SUBAPPLICATION Uebung_016 (* Subapplication Type *)
  (* Standard: 61499-2 *)
  (* Version 1.0, 2023-10-23, franz *)
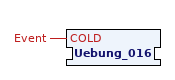
  EVENT_INPUT
    COLD;
  END_EVENT
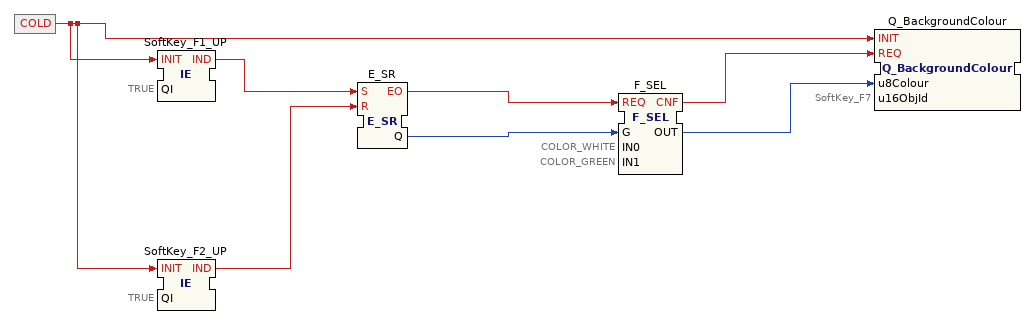
  FBS
    SoftKey_F1_UP : IE(QI := TRUE);
    SoftKey_F2_UP : IE(QI := TRUE);
    E_SR : E_SR;
    F_SEL : F_SEL(IN0 := COLOR_WHITE, IN1 := COLOR_GREEN);
    Q_BackgroundColour : Q_BackgroundColour(u16ObjId := SoftKey_F7);
  END_FBS
  EVENT_CONNECTIONS
    COLD TO SoftKey_F1_UP.INIT;
    COLD TO SoftKey_F2_UP.INIT;
    SoftKey_F1_UP.IND TO E_SR.S;
    SoftKey_F2_UP.IND TO E_SR.R;
    E_SR.EO TO F_SEL.REQ;
    COLD TO Q_BackgroundColour.INIT;
    F_SEL.CNF TO Q_BackgroundColour.REQ;
  END_CONNECTIONS
  DATA_CONNECTIONS
    E_SR.Q TO F_SEL.G;
    F_SEL.OUT TO Q_BackgroundColour.u8Colour;
  END_CONNECTIONS
END_SUBAPPLICATION
